PROGRAM main
VAR
	Timer_Pause : TON;
	Timer_Lys : TON;
	TimerLysOn : bool;
	PresetTime : time := T#600ms;
	PresetTime1 : time := T#300ms;
	REDLed : bool;
END_VAR

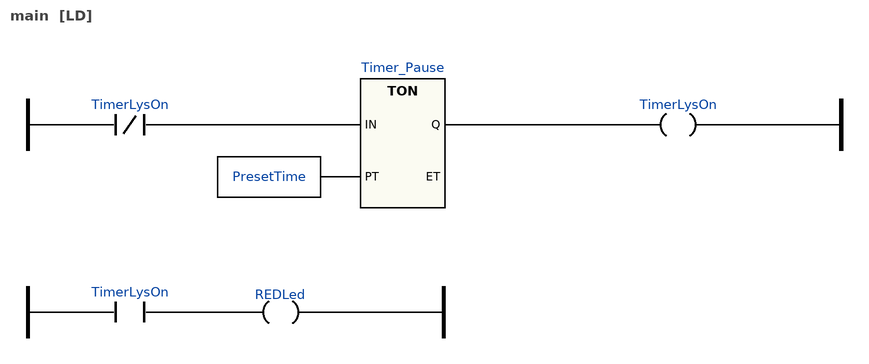
(* LD diagram, written out as Structured Text *)
Timer_Pause(IN := NOT TimerLysOn, PT := PresetTime);
TimerLysOn := Timer_Pause.Q;
REDLed := TimerLysOn;
END_PROGRAM
